TYPE "UDT_RecipeHeader"
VERSION : 0.1
   STRUCT
      ProductName : String[48];
      ProductID : String[48];
      RecipeVersion : String[18];
      FixtureFamily : Int;
      Enabled : Bool;
      CreatedBy : String[24];
      UpdatedBy : String[24];
      CreatedTS : Date_And_Time;
      UpdatedTS : Date_And_Time;
      Comment : String[96];
   END_STRUCT;

END_TYPE

